FUNCTION_BLOCK fb_prod_comp_ctrl

VAR_INPUT
	kc: REAL := 0.0;
	ti:REAL := 0.0;
	ts:REAL := 0.0;
	hi:REAL := 0.0;
	lo:REAL := 0.0;
	x0:REAL := 0.0;
	set_prod_rate: REAL := g_set_production;
	//xmv17: REAL;

END_VAR

VAR_OUTPUT
	Prodsp: REAL := 0;
	Fp: REAL :=0;
END_VAR

VAR
	
	pct_g_dpi: fb_discrete_pi := (kc := 0.4, ti := 100.0, ts := g_Ts_base, hi := 100, lo:=0.0);
	zoh_real_0: fb_zoh_real := (xlast := x0 );
	change_rate_limit: FB_CTRL_LIMITER := (stInternalParams := (fMinOutput := -0.286875, fMaxOutput := 0.286875));
	rate: REAL := 0;
	
	prodsp_scaled: REAL;
	calc_change_rate: FB_CTRL_D;
	integrate_change_rate: FB_CTRL_I;
	prod_rate_saturate: FB_CTRL_LIMITER;
	prod_rate_saturate_params: ST_CTRL_LIMITER_PARAMS := (fMinOutput := lo, fMaxOutput := hi);
	last_prod_rate: REAL := 0.0;
	
	stparams_calc_change_rate: ST_CTRL_D_PARAMS;
	stparams_change_rate_limit: ST_CTRL_LIMITER_PARAMS;
	stparams_integrate_change_rate: ST_CTRL_I_PARAMS;
	
	pctgsp: REAL := 0.0;
	
	
END_VAR

VAR CONSTANT
	ProdspGain: REAL := 100/22.89;
END_VAR

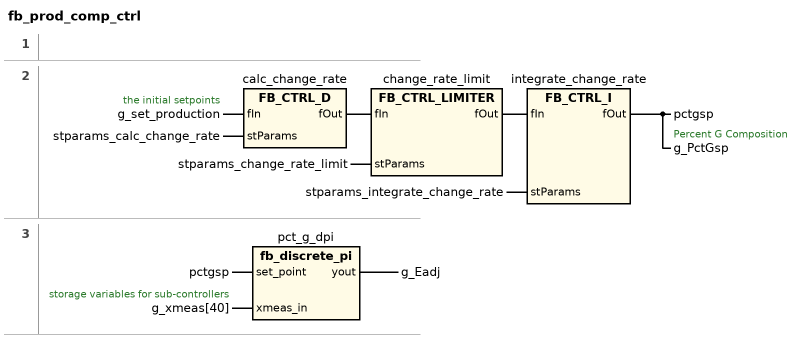
// NETWORK 1

// NETWORK 2
//   g_set_production: the initial setpoints
//   g_PctGsp: Percent G Composition
calc_change_rate(fIn := g_set_production, stParams := stparams_calc_change_rate); // FB_CTRL_D
change_rate_limit(fIn := calc_change_rate.fOut, stParams := stparams_change_rate_limit); // FB_CTRL_LIMITER
integrate_change_rate(fIn := change_rate_limit.fOut, stParams := stparams_integrate_change_rate); // FB_CTRL_I
pctgsp := integrate_change_rate.fOut;
g_PctGsp := integrate_change_rate.fOut;

// NETWORK 3
//   g_xmeas[40]: storage variables for sub-controllers
pct_g_dpi(set_point := pctgsp, xmeas_in := g_xmeas[40]); // fb_discrete_pi
g_Eadj := pct_g_dpi.yout;

END_FUNCTION_BLOCK

(* stored: Version 1.1.0.1, ProductVersion 3.1.0.26
   POU fb_prod_comp_ctrl: Id {b903bd3d-7f3b-4c5b-bdbb-2641db0bfa02} *)
